// TwinCAT 3 PLC project Untitled1
// ProgramVersion: 3.1.4023.0
// libraries:
//   Tc2_Standard, * (Beckhoff Automation GmbH)
//   Tc2_System, * (Beckhoff Automation GmbH)
//   Tc2_Utilities, * (Beckhoff Automation GmbH)
//   Tc3_Module, * (Beckhoff Automation GmbH)
// project tree:
//   / PlcTask.TcTTO
//   POUs/ MAIN.TcPOU
// real-time tasks:
//   TASK PlcTask: cycle T#10ms, priority 20, ADS port 350

CONFIGURATION Untitled1
    RESOURCE PLC ON TwinCAT3
        TASK PlcTask(INTERVAL := T#10ms, PRIORITY := 20);
        PROGRAM MAIN WITH PlcTask : MAIN;
    END_RESOURCE
END_CONFIGURATION

// ---- POUs/MAIN.TcPOU
PROGRAM MAIN
VAR
	bToggleFlashing : BOOL;
	nCounter: INT;
	bGaugeOn: BOOL;
	
	GaugeTimer: TON;
	GaugeTrig: R_TRIG;
	bGaugeTimerOn: BOOL;
	GaugeCounter: INT;
	
	fbGetLicenses : FB_GetLicensesEx;
	
	iWriteIntHere : INT;
	
END_VAR

nCounter := nCounter +1;

fbGetLicenses.bExecute := true;

IF bGaugeOn THEN
	GaugeTimer(IN:= bGaugeTimerOn, PT:=T#1S , Q=> , ET=> );
	IF GaugeTimer.Q THEN
		bGaugeTimerOn := FALSE;
		GaugeTrig(CLK:= bGaugeOn, Q=> );
		IF GaugeTrig.Q THEN
			GaugeCounter := GaugeCounter + 1;
			bGaugeOn := FALSE;
		END_IF
	END_IF
END_IF

END_PROGRAM
